FUNCTION F_LogWarning : T_MaxString 
VAR_INPUT
    Message : T_MaxString;
END_VAR

ADSLOGSTR(
    msgCtrlMask := ADSLOG_MSGTYPE_STRING OR ADSLOG_MSGTYPE_WARN OR ADSLOG_MSGTYPE_LOG,
    msgFmtStr := Message,
    strArg := '');

END_FUNCTION

(* stored: Version 1.1.0.1, ProductVersion 3.1.4024.3
   POU F_LogWarning: Id {3b935c52-6ca0-4698-a6d8-fa6889a094b4}, SpecialFunc None *)
